TYPE stDIGDiagInput :
STRUCT
	{attribute addProperty Name "Overtemperature"}
	Overtemperature AT %I* : BIT;
	{attribute addProperty Name "Open Load"}
	OpenLoad AT %I* : BIT;
	{attribute addProperty Name "Overcurrent"}
	Overcurrent AT %I* : BIT;
	{attribute addProperty Name "Short Circuit to 24V"}
	ShortCircuitTo24V AT %I* : BIT;
END_STRUCT
END_TYPE

(* stored: Version 1.1.0.1, ProductVersion 3.1.4024.9
   DUT stDIGDiagInput: Id {16e39790-9865-0db8-3a9b-f3baffcea9c6} *)
